# B&R Automation Studio project TrkMster
Automation Studio 4.7.5.60 SP; technology packages: mappMotion 5.12.0, mappView 5.12.0

## Configuration Config1

CPU PC_any, AutomationRuntime C4.72, Build 6.3.0, Safety 0.0, Vc V4.72.0

### Task classes (Cpu.sw)
```
Cyclic#1 (cycle 800 us, tolerance 1600 us):
  TrakMain <- Source.Trak.TrakMain.prg
Cyclic#4:
  Version <- Source.Support.Version.Version.prg
  MachineInf <- Source.Support.MachineInfo.prg
Cyclic#8 (cycle 800 us):
  Program <- Source.Program.prg
DataObjects: McAcpSys
Binaries: FWRules, McAcpSim, arcoal, arsvcreg, TCData, McAcpDrv, mvLoader, arflatprv, udbdef, iomap, Config_1, arconfig, asfw, ashwac, sysconf, User, Role, ashwd, Config_2
Libraries: AsBrStr, McBase, McAxis, McAcpTrak, MpBase, powerlnk, asieccon, sys_lib, arssl, TrkMst, snprintf, LoggingLib, astime, runtime, asstring, ArEventLog, AsTCP, FileIO, brdkSTR
```

### Hardware
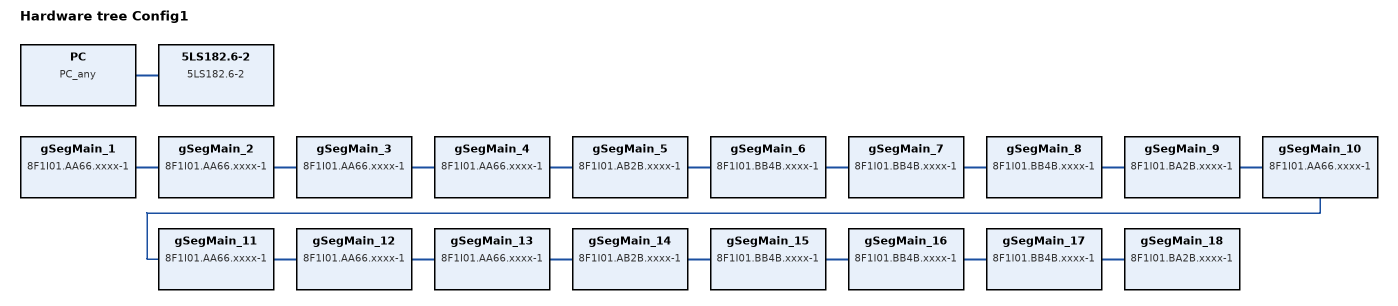
```
5LS182.6-2 : 5LS182.6-2 v1.7.0.0  [SL -> PC.SL1]
PC : PC_any v1.1.0.0 (OrderNumber=PC)
  ConfigurationID = TrkMster_Config1
  ConfigVersion = 0.0.1
  ConfigVersion = 0.1
  ConfigVersion = 0.1
  ConfigVersion = 0.1
  ConfigVersion = 0.1
  ConfigVersion = 0.1
  ConfigVersion = 0.1
  SystemTick = 800
  Cyclic1Duration = 800
  Cyclic1Tolerance = 1600
  Cyclic8Duration = 800
  FileDevice1
  FileDeviceName1 = SvgData
  FileDevicePath1 = ../../../../Logical/SceneViewer/Generated
  ActivateOpcUa = 1
  OpcUaInformationModels_PV_Version = 1
gSegMain_1 : 8F1I01.AA66.xxxx-1 v1.0.0.2  [PLK2 -> gSegMain_2.PLK1 (NodeNumber=1) [Cable Type=PowerlinkCable, Length=10, Version=1.0.0.3]; PLK3 -> 5LS182.6-2.IF1 (NodeNumber=1) [Cable Type=PowerlinkCable, Length=10, Version=1.0.0.3]]
  DriveConfiguration:
    McTypeID = LLMConfig
  DriveConfiguration/Segment:
    Shape = STRAIGHT660
    SegmentReference = gSegMain_1
    StopReaction = UseAssemblySetting
    SpeedFilter = UseAssemblySetting
gSegMain_10 : 8F1I01.AA66.xxxx-1 v1.0.0.2  [PLK1 -> gSegMain_9.PLK2 [Cable Type=PowerlinkCable, Length=10, Version=1.0.0.3]; PLK2 -> gSegMain_11.PLK1 [Cable Type=PowerlinkCable, Length=10, Version=1.0.0.3]]
  DriveConfiguration:
    McTypeID = LLMConfig
  DriveConfiguration/Segment:
    Shape = STRAIGHT660
    SegmentReference = gSegMain_10
    StopReaction = UseAssemblySetting
    SpeedFilter = UseAssemblySetting
gSegMain_11 : 8F1I01.AA66.xxxx-1 v1.0.0.2  [PLK1 -> gSegMain_10.PLK2 [Cable Type=PowerlinkCable, Length=10, Version=1.0.0.3]; PLK2 -> gSegMain_12.PLK1 [Cable Type=PowerlinkCable, Length=10, Version=1.0.0.3]]
  DriveConfiguration:
    McTypeID = LLMConfig
  DriveConfiguration/Segment:
    Shape = STRAIGHT660
    SegmentReference = gSegMain_11
    StopReaction = UseAssemblySetting
    SpeedFilter = UseAssemblySetting
gSegMain_12 : 8F1I01.AA66.xxxx-1 v1.0.0.2  [PLK1 -> gSegMain_11.PLK2 [Cable Type=PowerlinkCable, Length=10, Version=1.0.0.3]; PLK2 -> gSegMain_13.PLK1 [Cable Type=PowerlinkCable, Length=10, Version=1.0.0.3]]
  DriveConfiguration:
    McTypeID = LLMConfig
  DriveConfiguration/Segment:
    Shape = STRAIGHT660
    SegmentReference = gSegMain_12
    StopReaction = UseAssemblySetting
    SpeedFilter = UseAssemblySetting
gSegMain_13 : 8F1I01.AA66.xxxx-1 v1.0.0.2  [PLK1 -> gSegMain_12.PLK2 [Cable Type=PowerlinkCable, Length=10, Version=1.0.0.3]; PLK2 -> gSegMain_14.PLK1 [Cable Type=PowerlinkCable, Length=10, Version=1.0.0.3]]
  DriveConfiguration:
    McTypeID = LLMConfig
  DriveConfiguration/Segment:
    Shape = STRAIGHT660
    SegmentReference = gSegMain_13
    StopReaction = UseAssemblySetting
    SpeedFilter = UseAssemblySetting
gSegMain_14 : 8F1I01.AB2B.xxxx-1 v1.0.0.2  [PLK1 -> gSegMain_13.PLK2 [Cable Type=PowerlinkCable, Length=10, Version=1.0.0.3]; PLK2 -> gSegMain_15.PLK1 [Cable Type=PowerlinkCable, Length=10, Version=1.0.0.3]]
  DriveConfiguration:
    McTypeID = LLMConfig
  DriveConfiguration/Segment:
    Shape = STRAIGHT105_TO_CIRCULAR
    SegmentReference = gSegMain_14
    StopReaction = UseAssemblySetting
    SpeedFilter = UseAssemblySetting
gSegMain_15 : 8F1I01.BB4B.xxxx-1 v1.0.0.2  [PLK1 -> gSegMain_14.PLK2 [Cable Type=PowerlinkCable, Length=10, Version=1.0.0.3]; PLK2 -> gSegMain_16.PLK1 [Cable Type=PowerlinkCable, Length=10, Version=1.0.0.3]]
  DriveConfiguration:
    McTypeID = LLMConfig
  DriveConfiguration/Segment:
    Shape = CIRCULAR
    SegmentReference = gSegMain_15
    StopReaction = UseAssemblySetting
    SpeedFilter = UseAssemblySetting
gSegMain_16 : 8F1I01.BB4B.xxxx-1 v1.0.0.2  [PLK1 -> gSegMain_15.PLK2 [Cable Type=PowerlinkCable, Length=10, Version=1.0.0.3]; PLK2 -> gSegMain_17.PLK1 [Cable Type=PowerlinkCable, Length=10, Version=1.0.0.3]]
  DriveConfiguration:
    McTypeID = LLMConfig
  DriveConfiguration/Segment:
    Shape = CIRCULAR
    SegmentReference = gSegMain_16
    StopReaction = UseAssemblySetting
    SpeedFilter = UseAssemblySetting
gSegMain_17 : 8F1I01.BB4B.xxxx-1 v1.0.0.2  [PLK1 -> gSegMain_16.PLK2 [Cable Type=PowerlinkCable, Length=10, Version=1.0.0.3]; PLK2 -> gSegMain_18.PLK1 [Cable Type=PowerlinkCable, Length=10, Version=1.0.0.3]]
  DriveConfiguration:
    McTypeID = LLMConfig
  DriveConfiguration/Segment:
    Shape = CIRCULAR
    SegmentReference = gSegMain_17
    StopReaction = UseAssemblySetting
    SpeedFilter = UseAssemblySetting
gSegMain_18 : 8F1I01.BA2B.xxxx-1 v1.0.0.2  [PLK1 -> gSegMain_17.PLK2 [Cable Type=PowerlinkCable, Length=10, Version=1.0.0.3]]
  DriveConfiguration:
    McTypeID = LLMConfig
  DriveConfiguration/Segment:
    Shape = CIRCULAR_TO_STRAIGHT105
    SegmentReference = gSegMain_18
    StopReaction = UseAssemblySetting
    SpeedFilter = UseAssemblySetting
gSegMain_2 : 8F1I01.AA66.xxxx-1 v1.0.0.2  [PLK1 -> gSegMain_1.PLK2 [Cable Type=PowerlinkCable, Length=10, Version=1.0.0.3]; PLK2 -> gSegMain_3.PLK1 [Cable Type=PowerlinkCable, Length=10, Version=1.0.0.3]]
  DriveConfiguration:
    McTypeID = LLMConfig
  DriveConfiguration/Segment:
    Shape = STRAIGHT660
    SegmentReference = gSegMain_2
    StopReaction = UseAssemblySetting
    SpeedFilter = UseAssemblySetting
gSegMain_3 : 8F1I01.AA66.xxxx-1 v1.0.0.2  [PLK1 -> gSegMain_2.PLK2 [Cable Type=PowerlinkCable, Length=10, Version=1.0.0.3]; PLK2 -> gSegMain_4.PLK1 [Cable Type=PowerlinkCable, Length=10, Version=1.0.0.3]]
  DriveConfiguration:
    McTypeID = LLMConfig
  DriveConfiguration/Segment:
    Shape = STRAIGHT660
    SegmentReference = gSegMain_3
    StopReaction = UseAssemblySetting
    SpeedFilter = UseAssemblySetting
gSegMain_4 : 8F1I01.AA66.xxxx-1 v1.0.0.2  [PLK1 -> gSegMain_3.PLK2 [Cable Type=PowerlinkCable, Length=10, Version=1.0.0.3]; PLK2 -> gSegMain_5.PLK1 [Cable Type=PowerlinkCable, Length=10, Version=1.0.0.3]]
  DriveConfiguration:
    McTypeID = LLMConfig
  DriveConfiguration/Segment:
    Shape = STRAIGHT660
    SegmentReference = gSegMain_4
    StopReaction = UseAssemblySetting
    SpeedFilter = UseAssemblySetting
gSegMain_5 : 8F1I01.AB2B.xxxx-1 v1.0.0.2  [PLK1 -> gSegMain_4.PLK2 [Cable Type=PowerlinkCable, Length=10, Version=1.0.0.3]; PLK2 -> gSegMain_6.PLK1 [Cable Type=PowerlinkCable, Length=10, Version=1.0.0.3]]
  DriveConfiguration:
    McTypeID = LLMConfig
  DriveConfiguration/Segment:
    Shape = STRAIGHT105_TO_CIRCULAR
    SegmentReference = gSegMain_5
    StopReaction = UseAssemblySetting
    SpeedFilter = UseAssemblySetting
gSegMain_6 : 8F1I01.BB4B.xxxx-1 v1.0.0.2  [PLK1 -> gSegMain_5.PLK2 [Cable Type=PowerlinkCable, Length=10, Version=1.0.0.3]; PLK2 -> gSegMain_7.PLK1 [Cable Type=PowerlinkCable, Length=10, Version=1.0.0.3]]
  DriveConfiguration:
    McTypeID = LLMConfig
  DriveConfiguration/Segment:
    Shape = CIRCULAR
    SegmentReference = gSegMain_6
    StopReaction = UseAssemblySetting
    SpeedFilter = UseAssemblySetting
gSegMain_7 : 8F1I01.BB4B.xxxx-1 v1.0.0.2  [PLK1 -> gSegMain_6.PLK2 [Cable Type=PowerlinkCable, Length=10, Version=1.0.0.3]; PLK2 -> gSegMain_8.PLK1 [Cable Type=PowerlinkCable, Length=10, Version=1.0.0.3]]
  DriveConfiguration:
    McTypeID = LLMConfig
  DriveConfiguration/Segment:
    Shape = CIRCULAR
    SegmentReference = gSegMain_7
    StopReaction = UseAssemblySetting
    SpeedFilter = UseAssemblySetting
gSegMain_8 : 8F1I01.BB4B.xxxx-1 v1.0.0.2  [PLK1 -> gSegMain_7.PLK2 [Cable Type=PowerlinkCable, Length=10, Version=1.0.0.3]; PLK2 -> gSegMain_9.PLK1 [Cable Type=PowerlinkCable, Length=10, Version=1.0.0.3]]
  DriveConfiguration:
    McTypeID = LLMConfig
  DriveConfiguration/Segment:
    Shape = CIRCULAR
    SegmentReference = gSegMain_8
    StopReaction = UseAssemblySetting
    SpeedFilter = UseAssemblySetting
gSegMain_9 : 8F1I01.BA2B.xxxx-1 v1.0.0.2  [PLK1 -> gSegMain_8.PLK2 [Cable Type=PowerlinkCable, Length=10, Version=1.0.0.3]; PLK2 -> gSegMain_10.PLK1 [Cable Type=PowerlinkCable, Length=10, Version=1.0.0.3]]
  DriveConfiguration:
    McTypeID = LLMConfig
  DriveConfiguration/Segment:
    Shape = CIRCULAR_TO_STRAIGHT105
    SegmentReference = gSegMain_9
    StopReaction = UseAssemblySetting
    SpeedFilter = UseAssemblySetting
```

### Config_1.assembly - PC/mappMotion/Config_1.assembly
```
Element gAssembly_1 (Type=assembly)
  Tracks:
    TrackSeparation = 0.030
    Track[1]:
      Segments:
        SegmentRef[1] = ::gSegMain_1
        SegmentRef[2] = ::gSegMain_2
        SegmentRef[3] = ::gSegMain_3
        SegmentRef[4] = ::gSegMain_4
        SegmentRef[5] = ::gSegMain_5
        SegmentRef[6] = ::gSegMain_6
        SegmentRef[7] = ::gSegMain_7
        SegmentRef[8] = ::gSegMain_8
        SegmentRef[9] = ::gSegMain_9
        SegmentRef[10] = ::gSegMain_10
        SegmentRef[11] = ::gSegMain_11
        SegmentRef[12] = ::gSegMain_12
        SegmentRef[13] = ::gSegMain_13
        SegmentRef[14] = ::gSegMain_14
        SegmentRef[15] = ::gSegMain_15
        SegmentRef[16] = ::gSegMain_16
        SegmentRef[17] = ::gSegMain_17
        SegmentRef[18] = ::gSegMain_18
      Position = Absolute
        SegmentRef = ::gSegMain_1
        SegmentCountDirection = RightToLeft
        Translation:
          X = 0.0
          Y = 0.0
          Z = 0.0
        Orientation:
          Angle1 = 0.0
          Angle2 = 0.0
          Angle3 = 0.0
  CommonSegmentSettings:
    SegmentSimulationOnPLC = Off
    StopReaction = InductionHalt
    SpeedFilter = NotUsed
    ControllerParameters:
      DefaultParameter:
        Controller:
          Position:
            ProportionalGain = 0.0
          Speed:
            ProportionalGain = 0.0
            IntegrationTime = 0.0
          FeedForward:
            TotalMass = 0.0
            ForcePositive = 0.0
            ForceNegative = 0.0
            SpeedForceFactor = 0.0
            ForceLoad = 0.0
        MovementErrorLimits:
          PositionError = 0.0
          VelocityError = 0.0
      AdditionalParameterSets = NotUsed
    ShuttleIdentificationTime = 0
  Shuttles:
    MaxShuttleCount = 10
    DistanceReserve:
      Collision = 0.002
      ErrorStop = 0.006
    ShuttleStereotypes:
      ShuttleStRef[1] = ShuttleStereotype_1
    MagnetPlateConfigurations:
      ShuttleType[1] = 8F1SA.100.xxxxxx-x
    CollisionAvoidance:
      Strategy = Constant
      MaximumModelDimensions:
        Length:
          ExtentToFront = 0.025
          ExtentToBack = 0.025
        Width:
          Width = 0.046
  Visualization:
    MonitoringPv = ::gShuttleMon
    ProcessingTaskClass = 1
```

### Config_2.shuttlestereotype - PC/mappMotion/Config_2.shuttlestereotype
```
Element ShuttleStereotype_1 (Type=shuttlestereotype)
  MeasurementUnit = 5067858
  MeasurementResolution = 0.00001
  MovementLimits = Internal
    VelocityIsReadOnly = 0
    Velocity:
      Velocity = 4.0
    AccelerationIsReadOnly = 0
    Acceleration:
      Acceleration = 10.0
    DecelerationIsReadOnly = 0
    Deceleration:
      Deceleration = 10.0
  JerkFilter = Used
    JerkTime = 0.02
  UserData:
    Size = 3
```

### Config_3.sector - PC/mappMotion/Config_3.sector
```
Element secMain (Type=sector)
  Type = Composed
    StartSegment:
      SegmentRef = ::gSegMain_1
    IntermediateSegments:
      SegmentRef[1] = ::gSegMain_2
      SegmentRef[2] = ::gSegMain_3
      SegmentRef[3] = ::gSegMain_4
      SegmentRef[4] = ::gSegMain_5
      SegmentRef[5] = ::gSegMain_6
      SegmentRef[6] = ::gSegMain_7
      SegmentRef[7] = ::gSegMain_8
      SegmentRef[8] = ::gSegMain_9
      SegmentRef[9] = ::gSegMain_10
      SegmentRef[10] = ::gSegMain_11
      SegmentRef[11] = ::gSegMain_12
      SegmentRef[12] = ::gSegMain_13
      SegmentRef[13] = ::gSegMain_14
      SegmentRef[14] = ::gSegMain_15
      SegmentRef[15] = ::gSegMain_16
      SegmentRef[16] = ::gSegMain_17
    EndSegment:
      SegmentRef = ::gSegMain_18
      PositionRelativeTo = FromEnd
```

## Logical view

Binary libraries used (declarations not repeated): operator, runtime, astime, AsIecCon, AsBrStr, McBase 5.12.0, McAxis 5.12.0, McAcpTrak 5.12.0, MpBase 5.12.0, snprintf 1.10.2, LoggingLib 2.30.1, asstring, ArEventLog, AsTCP, FileIO

### Global.typ - Global data types
```iecst
TYPE
	UserDataTyp : 	STRUCT
		Red : USINT;
		Green : USINT;
		Blue : USINT;
	END_STRUCT;
END_TYPE
```

### Global.var - Global variables
```iecst
VAR
	gShuttleMon : McAcpTrakAssemblyMonData;
	gPowered : BOOL;
END_VAR
```

### Segments.var - Global variables
```iecst
VAR
	gSegMain_1 : McSegmentType;
	gSegMain_2 : McSegmentType;
	gSegMain_3 : McSegmentType;
	gSegMain_4 : McSegmentType;
	gSegMain_5 : McSegmentType;
	gSegMain_6 : McSegmentType;
	gSegMain_7 : McSegmentType;
	gSegMain_8 : McSegmentType;
	gSegMain_9 : McSegmentType;
	gSegMain_10 : McSegmentType;
	gSegMain_11 : McSegmentType;
	gSegMain_12 : McSegmentType;
	gSegMain_13 : McSegmentType;
	gSegMain_14 : McSegmentType;
	gSegMain_15 : McSegmentType;
	gSegMain_16 : McSegmentType;
	gSegMain_17 : McSegmentType;
END_VAR
```

### Package Logical/Libraries - Global libraries

- Library Logical/Libraries/brdkSTR (ANSIC, version 1.03.1) (no source held here)

### Library Logical/Libraries/TrkMst (ANSIC)
Depends on: McAcpTrak, snprintf, brdkSTR

#### Types.typ - Exported data types
```iecst
(*Track Master Core Types*)

TYPE
	tmCoreInternalTyp : 	STRUCT  (*Internal Datatype*)
		TypeID : UDINT; (*TypeID to help with handle application*)
		State : USINT; (*State of execution*)
		Axes : ARRAY[0..tmMAX_SHUTLE_ARRAY]OF tmCoreAxisLookupTyp; (*Axis Lookup table based on the current Shuttle Index*)
		Fbs : tmCoreFbTyps; (*Internal Function blocks*)
		ShCount : USINT; (*Shuttle Count*)
	END_STRUCT;
	tmCoreViewBoxCfgTyp : 	STRUCT  (*Attributes of the SVG's viewbox*)
		MinX : REAL; (*Minimum x position*)
		MinY : REAL; (*minimum y position*)
		Width : REAL; (*Width of viewbox*)
		Height : REAL; (*Height of viewbox*)
	END_STRUCT;
	tmCoreStateEnum :
		( (*State of execution*)
		tmCORE_OFF, (*Waiting for enable command*)
		tmCORE_INIT, (*Initialization state*)
		tmCORE_GET_SH, (*Get the shuttle in the assembly*)
		tmCORE_GET_NEXT, (*Set the next command*)
		tmCORE_RUNNING, (*Running state*)
		tmCORE_RESET, (*Resetting state*)
		tmCORE_ERROR (*Error state*)
		);
	tmCoreErrorEnum :
		( (*Error Enumeration*)
		tmCORE_ERR_OK := 0, (*No error present*)
		tmCORE_ERR_INVALID_ASSEMBLY := -61000, (*Invalid input assembly reference*)
		tmCORE_ERR_SH_COUNT_EXCEEDED := -61001, (*Maximum shuttle count exceeded. Need to increase max shuttle count constant*)
		tmCORE_ERR_STR_LEN_EXCEEDED := -61002 (*The built string is too long, need to increase the maximum size to prevent page faulting*)
		);
	tmCoreSvgLengthsTyp : 	STRUCT  (*String lengths of SVGs*)
		ContentLength : UDINT; (*String Length of SVG Content string*)
		TransformLength : UDINT; (*String Length of SVG Transform string*)
	END_STRUCT;
	tmCoreFbTyps : 	STRUCT  (*Internal Function blocks*)
		AsmGetShuttle : MC_BR_AsmGetShuttle_AcpTrak;
	END_STRUCT;
	tmCoreAxisLookupTyp : 	STRUCT  (*Lookup table datatype*)
		Present : BOOL; (*Axis is present and a valid reference exists*)
		Axis : McAxisType; (*Axis information*)
	END_STRUCT;
	tmCoreOptionsTyp : 	STRUCT  (*Options for Core Function Block*)
		Color : tmCoreColorOptionTyp; (*Shuttle Color Option*)
	END_STRUCT;
	tmCoreColorOptionTyp : 	STRUCT  (*Shuttle Color Option*)
		Enabled : BOOL; (*Option is enabled*)
		Offsets : tmCoreColorOffsetsTyp; (*Userdata color offsets*)
	END_STRUCT;
	tmCoreColorOffsetsTyp : 	STRUCT  (*Userdata color offsets*)
		Red : UDINT; (*Offset for UserData address for the Red color in USINT*)
		Green : UDINT; (*Offset for UserData address for the Green color in USINT*)
		Blue : UDINT; (*Offset for UserData address for the Blue color in USINT*)
	END_STRUCT;
END_TYPE

(*Track Master Shuttle Control Types*)

TYPE
	tmShuttleControlParsTyp : 	STRUCT  (*Input parameters for Shuttle Control*)
		Position : LREAL; (*Destination position for Absolute and Velocity commands*)
		Distance : LREAL; (*Distance for all relative commands*)
		Vel : REAL; (*Comanded Movement velocity*)
		Accel : REAL; (*Comanded Movement acceleration*)
		Decel : REAL; (*Comanded Movement deceleration*)
	END_STRUCT;
	tmShuttleControlInternalTyp : 	STRUCT  (*Internal data type*)
		State : tmShuttleControlStatesEnum; (*State of execution*)
		CoreInt : REFERENCE TO tmCoreInternalTyp; (*Internal data for the Core function block*)
		CurrentAxis : McAxisType; (*Current selected Axis*)
		Fbs : tmShuttleControlFbTyp; (*Internal function blocks*)
		Idx : USINT; (*Selected Index for the axis lookup table*)
		LastIdx : USINT; (*Last cycle selected index for the axis lookup table*)
	END_STRUCT;
	tmShuttleControlFbTyp : 	STRUCT  (*Internal Function Blocks*)
		ShGetInfo : MC_BR_ShReadInfo_AcpTrak; (*Shuttle Get info*)
		ElMoveAbs : MC_BR_ElasticMoveAbs_AcpTrak; (*Elastic move absolute command*)
		ElMoveAdd : MC_BR_ElasticMoveAdd_AcpTrak; (*Elastic move addtive command*)
	END_STRUCT;
	tmShuttleControlErrorEnum :
		( (*Error enumeration*)
		tmSH_CONTROL_ERR_OK := 0, (*No error currently*)
		tmSH_CONTROL_WARN_SH_NOT_AVAIL := -52000, (*Shuttle Currently not listed as available*)
		tmSH_CONTROL_WARN_NO_ELEM_FND := -52001, (*Input selected element did not return a shuttle*)
		tmSH_CONTROL_ERR_INVALID_HANDLE := -62000, (*Invalid input handle*)
		tmSH_CONTROL_ERR_EL_MOVE := -62001 (*Error in an elastic movment*)
		);
	tmShuttleControlStatesEnum :
		( (*State of execution*)
		tmSH_CONTROL_OFF, (*Off State*)
		tmSH_CONTROL_INIT, (*Init/Waiting for valid ShElement state*)
		tmSH_CONTROL_IDLE, (*Idle waiting for a command state*)
		tmSH_CONTROL_EL_MOVE_ABS, (*Move Elastic absoulte active state*)
		tmSH_CONTROL_EL_MOVE_ADD, (*Move Elastic Additive active state*)
		tmSH_CONTROL_MOVE_DONE, (*Move has completed*)
		tmSH_CONTROL_ERROR (*Error present on the FB*)
		);
END_TYPE
```

#### Constants.var - Exported constants
```iecst
VAR CONSTANT
	tmMAX_SHUTTLE_COUNT : USINT := 150;
	tmMAX_SHUTLE_ARRAY : USINT := tmMAX_SHUTTLE_COUNT-1;
	tmCORE_CORE_TYPE_ID : DINT := 651684313;
	tmCORE_MAX_STR_LEN : UDINT := 3000;
END_VAR
```

#### TrkMst.fun - Exported functions and function blocks
```iecst
FUNCTION_BLOCK tmCore (*Core Track Master Function Block*)
	VAR_INPUT
		Enable : BOOL; (*Enables the core functionality*)
		ErrorRest : BOOL; (*Reset any present errors*)
		Assembly : REFERENCE TO McAssemblyType; (*Assembly reference to monitor*)
		ShuttleMon : REFERENCE TO McAcpTrakAssemblyMonData; (*Shuttle Monitor structure for the assembly*)
		ViewBoxCfg : tmCoreViewBoxCfgTyp; (*View box configuration for the SVG*)
		Options : REFERENCE TO tmCoreOptionsTyp; (*Options for the core fb*)
	END_VAR
	VAR_OUTPUT
		Error : BOOL; (*Error present on FB*)
		ErrorID : tmCoreErrorEnum; (*Error ID of current error*)
		Active : BOOL; (*Function block is active*)
		SvgContent : STRING[tmCORE_MAX_STR_LEN]; (*SVG Content string to tie to a Paper widget*)
		SvgTransform : STRING[tmCORE_MAX_STR_LEN]; (*SVG Transform string to tie to a paper widget*)
		StrLengths : tmCoreSvgLengthsTyp; (*Diagnostic viewer to see current lengths of SVG Content/Transform*)
		Handle : UDINT; (*Handle used for other Track Master Function Blocks*)
	END_VAR
	VAR
		Internal : tmCoreInternalTyp; (*Internal data type*)
	END_VAR
END_FUNCTION_BLOCK

FUNCTION_BLOCK tmShuttleControl (*Shuttle Control Function Block*)
	VAR_INPUT
		Enable : BOOL; (*Enables the shuttle controller*)
		Handle : UDINT; (*Handle of the Core Track Master Function Block*)
		SelectedElem : STRING[80]; (*Selected Element String that is populated from a Paper Widget*)
		ElasticMoveAbs : BOOL; (*Command to send shuttle on Elastic Move Absolute*)
		ElasticMoveAdd : BOOL; (*Command to send shuttle on Elastic Move Additive*)
		Parameters : REFERENCE TO tmShuttleControlParsTyp; (*Parameters for movement commands*)
	END_VAR
	VAR_OUTPUT
		Active : BOOL; (*Function block is currently Active*)
		MovementActive : BOOL; (*Controlled Shuttle is currently moving*)
		MovementDone : BOOL; (*Controlled Shuttle has completed movement*)
		Valid : BOOL; (*Input Selected Element is a valid controllable shuttle*)
		ShInfo : McAcpTrakShInfoType; (*Selected shuttle's current info. Only is Valid when Valid flag is set*)
		Error : BOOL; (*Error Present on FB*)
		ErrorID : DINT; (*Error ID of current Error*)
	END_VAR
	VAR
		Internal : tmShuttleControlInternalTyp; (*Internal data type*)
	END_VAR
END_FUNCTION_BLOCK
```

#### tmCore.c
```c
#include <bur/plctypes.h>

#define TRUE 1
#define FALSE 0

#ifdef __cplusplus
	extern "C"
	{
#endif
#include "TrkMst.h"
#ifdef __cplusplus
	};
#endif
//Verify that the two string lengths do not exceed a length
plcbit CheckStrLen(char* dest,char* source,UDINT length){
	if(brdkStrLen(dest) + brdkStrLen(source) >= length){
		return FALSE;
	}
	else{
		return TRUE;
	}
}
DINT BuildShuttlePolygon(char* dest,
		USINT idx,
		LREAL length,
		LREAL width,
		UDINT userDataAdr,
		struct tmCoreColorOptionTyp* colorOption){

	char tmp[150];
	USINT red,blue,green;
	struct UserDataTyp* tst;

	if(!colorOption->Enabled){
		snprintf2(tmp,150,"<polygon id=\"sh%d\" points=\"0,0 %0f,0 , %f,%f %f,%f 0,%f\" style=\"fill:rgb(0,255,0);\"/>",
			idx,	//polygon index
			(length-width/2.0),//p1.x
			length,	//p1.y
			width/2.0, //p2.x
			(length-width/2.0),//p2.y
			width,//p2.x
			width); //p3.y
	}
	else{
		brsmemcpy(&red,userDataAdr + colorOption->Offsets.Red,sizeof(USINT));
		brsmemcpy(&green,userDataAdr + colorOption->Offsets.Green,sizeof(USINT));
		brsmemcpy(&blue,userDataAdr + colorOption->Offsets.Blue,sizeof(USINT));

		snprintf2(tmp,150,"<polygon id=\"sh%d\" points=\"0,0 %0f,0 , %f,%f %f,%f 0,%f\" style=\"fill:rgb(%d,%d,%d);\"/>",
			idx,	//polygon index
			(length-width/2.0),//p1.x
			length,	//p1.y
			width/2.0, //p2.x
			(length-width/2.0),//p2.y
			width,//p2.x
			width,
			red,
			green,
			blue); //p3.y
	}
	if(CheckStrLen(dest,&tmp,tmCORE_MAX_STR_LEN)){
		brsstrcat(dest,&tmp);
		return tmCORE_ERR_OK;
	}
	else
		return tmCORE_ERR_STR_LEN_EXCEEDED;
}

//This function loops through the assembly monitor data and builds a SVG string + SVG Transform. Will return 0 if succesful
//Will monitor to make sure the string lengths are not exceeded
DINT BuildStrings(struct McAcpTrakAssemblyMonData* mon,
		char* svgContent,char* svgTransform,
		struct tmCoreViewBoxCfgTyp* viewBox,
		struct tmCoreOptionsTyp* coreOptions){
	USINT i;
	USINT transCounter;
	transCounter = 0;
	char tmp[150];
	brsmemset(svgContent,0,sizeof(svgContent));
	brsmemset(svgTransform,0,sizeof(svgTransform));

	snprintf2(tmp,150,"<svg viewBox=\"%f %f %f %f\">",
		viewBox->MinX,
		viewBox->MinY,
		viewBox->Width,
		viewBox->Height);
	if(CheckStrLen(svgContent,&tmp,tmCORE_MAX_STR_LEN)){
		brsstrcat(svgContent,&tmp);
	}
	else
		return tmCORE_ERR_STR_LEN_EXCEEDED;
	brsstrcat(svgTransform,&"[");

	for (i = 0; i < tmMAX_SHUTTLE_COUNT; i++){
		if(mon->Shuttle[i].Available){
			brsmemset(&tmp,0,sizeof(tmp));

			LREAL width;
			LREAL length;
			LREAL shCenterX;
			LREAL shCenterY;

			width = mon->Shuttle[i].Width / 1000.0;
			length = (mon->Shuttle[i].ExtentToBack + mon->Shuttle[i].ExtentToFront)/ 1000.0;
			shCenterX = mon->Shuttle[i].Position.X / 1000.0 - mon->Shuttle[i].ExtentToBack / 1000.0;
			shCenterY = -(mon->Shuttle[i].Position.Y / 1000.0 + width / 2.0);

			snprintf2(tmp,150,"<g id=\"Shuttle%d\">",mon->Shuttle[i].Index);
			if(CheckStrLen(svgContent,&tmp,tmCORE_MAX_STR_LEN)){
				brsstrcat(svgContent,&tmp);
			}
			else
				return tmCORE_ERR_STR_LEN_EXCEEDED;

			DINT returnVal;
			returnVal = BuildShuttlePolygon(svgContent,mon->Shuttle[i].Index,length,width,mon->Shuttle[i].UserData,&coreOptions->Color);
			if(returnVal!= tmCORE_ERR_OK)
				return returnVal;

			snprintf2(tmp,150,"<text x=\"%f\" y=\"%f\" font-weight=\"bold\" font-size=\"0.035px\">%d</text>",
				mon->Shuttle[i].ExtentToBack / 2000.0,
				width * 3.0 / 4.0,
				mon->Shuttle[i].Index);
			if(CheckStrLen(svgContent,&tmp,tmCORE_MAX_STR_LEN)){
				brsstrcat(svgContent,&tmp);
			}
			else
				return tmCORE_ERR_STR_LEN_EXCEEDED;

			//Create an invisible bounding rectangle to handle the click event. "Invisible" by using the alpha channel, if you use the
			//Vibisility property, the click event will not fire for the SVG
			snprintf2(tmp,150,"<rect id=\"ID%d\" width=\"%f\" height=\"%f\" style=\"fill:rgba(0,0,0,0)\"/>",
				mon->Shuttle[i].Index,
				length,
				width);
			if(CheckStrLen(svgContent,&tmp,tmCORE_MAX_STR_LEN)){
				brsstrcat(svgContent,&tmp);
			}
			else
				return tmCORE_ERR_STR_LEN_EXCEEDED;

			if(CheckStrLen(svgContent,&"</g>",tmCORE_MAX_STR_LEN)){
				brsstrcat(svgContent,&"</g>");
			}
			else
				return tmCORE_ERR_STR_LEN_EXCEEDED;

			//Check to see if we've had more transforms to add a comma between the units
			if(transCounter>0){
				if(CheckStrLen(svgTransform,&",",tmCORE_MAX_STR_LEN)){
					brsstrcat(svgTransform,&",");
				}
				else
					return tmCORE_ERR_STR_LEN_EXCEEDED;
			}
			//Preform translation
			snprintf2(tmp,150,"{\"select\":\"#Shuttle%d\",\"duration\":100,\"display\":true,\"translate\":[%f,%f]},",
				mon->Shuttle[i].Index,
				shCenterX,
				shCenterY,
				-mon->Shuttle[i].Orientation.Angle1,
				length/2.0,
				width/2.0);
			if(CheckStrLen(svgTransform,&tmp,tmCORE_MAX_STR_LEN)){
				brsstrcat(svgTransform,&tmp);
			}
			else
				return tmCORE_ERR_STR_LEN_EXCEEDED;
			//Preform rotation
			snprintf2(tmp,150,"{\"select\":\"#sh%d\",\"duration\":100,\"display\":true,\"spin\":[%f,%f,%f]}",
				mon->Shuttle[i].Index,
				-mon->Shuttle[i].Orientation.Angle1, //Spin amount
				length/2.0,	//Spin center x
				width/2.0); //Spin center y
			if(CheckStrLen(svgTransform,&tmp,tmCORE_MAX_STR_LEN)){
				brsstrcat(svgTransform,&tmp);
			}
			else
				return tmCORE_ERR_STR_LEN_EXCEEDED;
			transCounter++;
		}

	}
	if(CheckStrLen(svgContent,&"</svg>",tmCORE_MAX_STR_LEN)){
		brsstrcat(svgContent,&"</svg>");
	}
	else
		return tmCORE_ERR_STR_LEN_EXCEEDED;
	if(CheckStrLen(svgTransform,&"]",tmCORE_MAX_STR_LEN)){
		brsstrcat(svgTransform,&"]");
	}
	else
		return tmCORE_ERR_STR_LEN_EXCEEDED;

	//No Error, finished everything return OK
	return tmCORE_ERR_OK;
}

/* Core Track Master function blocks. Handles the building of the SVG string */
void tmCore(struct tmCore* inst)
{
	switch (inst->Internal.State){
		case tmCORE_OFF:
			//******************************************************************************** Off state
			if(inst->Enable){
				inst->Internal.TypeID = tmCORE_CORE_TYPE_ID;
				inst->Handle = &inst->Internal;

				inst->Internal.Fbs.AsmGetShuttle.Assembly = inst->Assembly;
				inst->Internal.Fbs.AsmGetShuttle.Enable = TRUE;
				inst->Active = TRUE;
				inst->Internal.State = tmCORE_INIT;
			}
			break;
		case tmCORE_INIT:
			//Reset the lookup array just for safety
			brsmemset(&inst->Internal.Axes,0,sizeof(inst->Internal.Axes));

        	inst->Internal.State = tmCORE_GET_SH;
			break;
		case tmCORE_GET_SH:
			//******************************************************************************** Get Shuttle state
			if(inst->Internal.Fbs.AsmGetShuttle.Error){
				inst->Error = TRUE;
				inst->ErrorID = tmCORE_ERR_INVALID_ASSEMBLY;

				inst->Internal.State = tmCORE_ERROR;
			}
			else if(inst->Internal.Fbs.AsmGetShuttle.Valid){
				if(inst->Internal.Fbs.AsmGetShuttle.TotalCount >= tmMAX_SHUTTLE_COUNT
				|| inst->Internal.Fbs.AsmGetShuttle.AdditionalInfo.ShuttleID >= tmMAX_SHUTTLE_COUNT){

					inst->Error = TRUE;
					inst->ErrorID = tmCORE_ERR_SH_COUNT_EXCEEDED;

					inst->Internal.State = tmCORE_ERROR;
				}
				else{
					inst->Internal.Axes[inst->Internal.Fbs.AsmGetShuttle.AdditionalInfo.ShuttleID].Present = TRUE;
					inst->Internal.Axes[inst->Internal.Fbs.AsmGetShuttle.AdditionalInfo.ShuttleID].Axis = inst->Internal.Fbs.AsmGetShuttle.Axis;
					inst->Internal.Fbs.AsmGetShuttle.Next = FALSE;

					if(inst->Internal.Fbs.AsmGetShuttle.RemainingCount == 0){
						//Done populating the lookup array, moving on
						inst->Internal.Fbs.AsmGetShuttle.Enable = FALSE;

						inst->Internal.State = tmCORE_RUNNING;
					}
					else{
						inst->Internal.ShCount++;

						inst->Internal.State = tmCORE_GET_NEXT;
					}
				}
			}
			break;
		case tmCORE_GET_NEXT:
			//******************************************************************************** Get next shuttle state
			inst->Internal.Fbs.AsmGetShuttle.Next = TRUE;
			inst->Internal.State = tmCORE_GET_SH;
			break;
		case tmCORE_RUNNING:
			inst->ErrorID = BuildStrings(inst->ShuttleMon,&inst->SvgContent,&inst->SvgTransform,&inst->ViewBoxCfg,inst->Options);
			inst->StrLengths.ContentLength = brdkStrLen(&inst->SvgContent);
			inst->StrLengths.TransformLength = brdkStrLen(&inst->SvgTransform);

			if(inst->ErrorID != tmCORE_ERR_OK){
				inst->Error = TRUE;

				inst->Internal.State = tmCORE_ERROR;
			}
			break;
		case tmCORE_RESET:
        	//Try and recover by resetting any blocks

			break;
		case tmCORE_ERROR:
			if(inst->ErrorRest){
				inst->Error = FALSE;
				inst->ErrorID = tmCORE_ERR_OK;

				inst->Internal.State = tmCORE_OFF;
			}
			break;
	}
	//FB calls
	MC_BR_AsmGetShuttle_AcpTrak(&inst->Internal.Fbs.AsmGetShuttle);
}
```

#### tmShuttleControl.c
```c
#include <bur/plctypes.h>

#define TRUE 1
#define FALSE 0

#ifdef __cplusplus
	extern "C"
	{
#endif
#include "TrkMst.h"
#ifdef __cplusplus
	};
#endif

plcbit CheckValidity(char* selectedElem){
	char buf[2];
	//Get a substring of the first 3 characters
	brdkStrSubStr(&buf,selectedElem,0,3);
	//Look at the start of the selectedID, if it starts with #ID then we know a shuttle has been clicked
	if(0 == brsstrcmp(&buf,&"#ID")){
		return TRUE;
	}
	else{
		return FALSE;
	}
}
USINT GetIndex(char* selectedElem){
	char buf[3];
	brdkStrSubStr(&buf,selectedElem,3,brdkStrLen(selectedElem) - 3);
	return (USINT)brdkStrAToUdint(&buf,BRDK_STR_CONVERT_DECIMAL);
}
/* Function block for handling a shuttle control provided from the paper element's selected element ID. Must be paired with the tmCore FB */
void tmShuttleControl(struct tmShuttleControl* inst)
{
	if(inst->Valid){
		inst->ShInfo = inst->Internal.Fbs.ShGetInfo.ShuttleInfo;
	}
	switch (inst->Internal.State){
		case tmSH_CONTROL_OFF:
			//******************************************************************************** Off state
			if(inst->Enable){
				if(inst->Handle == 0){
					inst->Error = TRUE;
					inst->ErrorID = tmSH_CONTROL_ERR_INVALID_HANDLE;

					inst->Internal.State = tmSH_CONTROL_ERROR;
				}
				else{
					inst->Internal.CoreInt = (tmCoreInternalTyp*)inst->Handle;
					if(inst->Internal.CoreInt->TypeID != tmCORE_CORE_TYPE_ID){
						inst->Error = TRUE;
						inst->ErrorID = tmSH_CONTROL_ERR_INVALID_HANDLE;

						inst->Internal.State = tmSH_CONTROL_ERROR;
					}
					else{
						inst->Active = TRUE;

						inst->Internal.State = tmSH_CONTROL_INIT;
					}
				}
			}
			break;
		case tmSH_CONTROL_INIT:
			//******************************************************************************** Init state
			if(CheckValidity(&inst->SelectedElem)){	//Checking for the validity of the selected element format
				inst->Internal.Idx = GetIndex(&inst->SelectedElem);	//Pulling the index from the string
				if(inst->Internal.CoreInt->Axes[inst->Internal.Idx].Present){ //Verifying that index has a valid access in it
					inst->ErrorID = tmSH_CONTROL_ERR_OK;
					inst->Valid = TRUE;
					inst->Internal.CurrentAxis = inst->Internal.CoreInt->Axes[inst->Internal.Idx].Axis;

					inst->Internal.Fbs.ShGetInfo.Axis = &inst->Internal.CurrentAxis;
					inst->Internal.Fbs.ShGetInfo.Enable = TRUE;

					inst->Internal.State = tmSH_CONTROL_IDLE;
				}
				else{
					inst->ErrorID = tmSH_CONTROL_WARN_SH_NOT_AVAIL;
				}
			}
			else{
				inst->ErrorID = tmSH_CONTROL_WARN_NO_ELEM_FND;
			}

			break;
		case tmSH_CONTROL_IDLE:
			//******************************************************************************** Get Shuttle state
			//Need to check for if the selected element has changed
			inst->Internal.LastIdx = inst->Internal.Idx;
			if(CheckValidity(&inst->SelectedElem)){
				inst->Internal.Idx = GetIndex(&inst->SelectedElem);

				if(inst->Internal.Idx != inst->Internal.LastIdx){
					//We've changed indecies need to head back to init to reset the sh status
					inst->Valid = FALSE;
					inst->Internal.Fbs.ShGetInfo.Enable = FALSE;

					inst->Internal.State = tmSH_CONTROL_INIT;
				}
				else{
					//Here we can start parsing commands
					if(inst->ElasticMoveAbs){
						//Setup the elastic move absolute block and execute it
						inst->Internal.Fbs.ElMoveAbs.Axis = &inst->Internal.CurrentAxis;
						inst->Internal.Fbs.ElMoveAbs.Position = inst->Parameters->Position;
						inst->Internal.Fbs.ElMoveAbs.Velocity = inst->Parameters->Vel;
						inst->Internal.Fbs.ElMoveAbs.Acceleration = inst->Parameters->Accel;
						inst->Internal.Fbs.ElMoveAbs.Deceleration = inst->Parameters->Decel;

						inst->Internal.Fbs.ElMoveAbs.Execute = TRUE;

						inst->Internal.State = tmSH_CONTROL_EL_MOVE_ABS;
					}
					else if(inst->ElasticMoveAdd){
						//Setup the elastic move additve block and execute it
						inst->Internal.Fbs.ElMoveAdd.Axis = &inst->Internal.CurrentAxis;
						inst->Internal.Fbs.ElMoveAdd.Distance = inst->Parameters->Distance;
						inst->Internal.Fbs.ElMoveAdd.Velocity = inst->Parameters->Vel;
						inst->Internal.Fbs.ElMoveAdd.Acceleration = inst->Parameters->Accel;
						inst->Internal.Fbs.ElMoveAdd.Deceleration = inst->Parameters->Decel;

						inst->Internal.Fbs.ElMoveAdd.Execute = TRUE;

						inst->Internal.State = tmSH_CONTROL_EL_MOVE_ADD;
					}//End of commands check conditionals
				}
			}
			else{//We've received an invalid selection, need to reset the flags and Sh Status
				inst->Valid = FALSE;
				inst->Internal.Fbs.ShGetInfo.Enable = FALSE;

				inst->Internal.State = tmSH_CONTROL_INIT;
			}

			break;
		case tmSH_CONTROL_EL_MOVE_ABS:
			//******************************************************************************** Elastic Move absolute state
			if(inst->Internal.Fbs.ElMoveAbs.Error){
				inst->Error = TRUE;
				inst->ErrorID = tmSH_CONTROL_ERR_EL_MOVE;

				inst->Internal.State = tmSH_CONTROL_ERROR;
			}
			else if(inst->Internal.Fbs.ElMoveAbs.Active){
				inst->MovementActive = TRUE;
			}
			else if(inst->Internal.Fbs.ElMoveAbs.Done){
				inst->Internal.Fbs.ElMoveAbs.Execute = FALSE;
				inst->MovementActive = FALSE;
				inst->MovementDone = TRUE;

				inst->Internal.State = tmSH_CONTROL_MOVE_DONE;
			}
			break;
		case tmSH_CONTROL_EL_MOVE_ADD:
			//******************************************************************************** Elastic Move Additive state
			if(inst->Internal.Fbs.ElMoveAdd.Error){
				inst->Error = TRUE;
				inst->ErrorID = tmSH_CONTROL_ERR_EL_MOVE;

				inst->Internal.State = tmSH_CONTROL_ERROR;
			}
			else if(inst->Internal.Fbs.ElMoveAdd.Done){
				inst->MovementActive = FALSE;
				inst->MovementDone = TRUE;

				inst->Internal.Fbs.ElMoveAdd.Execute = FALSE;

				inst->Internal.State = tmSH_CONTROL_MOVE_DONE;
			}
			else{
				inst->MovementActive = TRUE;
			}
			break;
		case tmSH_CONTROL_MOVE_DONE:
			//******************************************************************************** Movement Done State
			if(!inst->ElasticMoveAbs
				&& !inst->ElasticMoveAdd){
				inst->MovementDone = FALSE;

				inst->Internal.State = tmSH_CONTROL_IDLE;
			}
			break;
		case tmSH_CONTROL_ERROR:
			//******************************************************************************** Error State
			if(!inst->Enable){
				inst->Error = FALSE;
				inst->ErrorID = tmSH_CONTROL_ERR_OK;

				inst->Internal.Fbs.ElMoveAbs.Execute = FALSE;
				inst->Internal.Fbs.ElMoveAdd.Execute = FALSE;
				inst->Internal.Fbs.ShGetInfo.Enable = FALSE;

				inst->Internal.Idx = 0;
				inst->Internal.LastIdx = 0;

				inst->Internal.State = tmSH_CONTROL_OFF;
			}
			break;
	}
	//FB calls

	MC_BR_ShReadInfo_AcpTrak(&inst->Internal.Fbs.ShGetInfo);
	MC_BR_ElasticMoveAbs_AcpTrak(&inst->Internal.Fbs.ElMoveAbs);
	MC_BR_ElasticMoveAdd_AcpTrak(&inst->Internal.Fbs.ElMoveAdd);
}
```

- Visualisation Logical/mappView (not shown)

### Program Logical/Source/TrackMaster (ANSIC)

#### Cyclic.c - Cyclic code
```c
/*********************************************************************************
 * Copyright: B&R Industrial Automation GmbH
 * Author:    trostelc
 * Created:   October 16, 2020/5:04 PM
 *********************************************************************************/

#include <bur/plctypes.h>

#ifdef _DEFAULT_INCLUDES
#include <AsDefault.h>
#endif

void _CYCLIC ProgramCyclic(void)
{
	//Build the SVG transform string
	//Start by adding the svg viewbox
	//Loop through the shuttle mon, if the shuttle is enabled, you'll take the X/Y/Z/rot and use it to build a <g> in the svg

	switch (state){
		case 0:
			if(start || gPowered){
				TrackMasterCore.Assembly = &gAssembly_1;
				TrackMasterCore.ShuttleMon = &gShuttleMon;
				TrackMasterCore.Enable = 1;

				//Set parameters for View box (this comes from the automatically generated SVG)
				TrackMasterCore.ViewBoxCfg.MinX = -3.37558;
				TrackMasterCore.ViewBoxCfg.MinY = -0.745;
				TrackMasterCore.ViewBoxCfg.Width = 4.11115;
				TrackMasterCore.ViewBoxCfg.Height = 0.86;

				state = 10;
			}
			break;
		case 10:
			if(TrackMasterCore.Active){
				ShControl.Enable = 1;
				ShControl.Handle = TrackMasterCore.Handle;
				ShControl.Parameters = &shPars;

				state = 20;
			}
			break;
		case 20:
			break;

	}

	brdkStrCpy(&ShControl.SelectedElem,&selectedId);

	tmCore(&TrackMasterCore);
	tmShuttleControl(&ShControl);

	//GetIndex();
}
```

#### Init.c - Initialization code
```c
#include <bur/plctypes.h>

#ifdef _DEFAULT_INCLUDES
	#include <AsDefault.h>
#endif

void _INIT ProgramInit(void)
{
	brsmemset(&selectedId,0,sizeof(selectedId));
	shPars.Accel = 10;
	shPars.Decel = 10;
	shPars.Vel = 1;
	coreOptions.Color.Enabled = 1;
	coreOptions.Color.Offsets.Red = 0;
	coreOptions.Color.Offsets.Green = 1;
	coreOptions.Color.Offsets.Blue = 2;
	TrackMasterCore.Options = &coreOptions;
}
```

#### Variables.var - Local variables
```iecst
VAR
	selectedId : STRING[80];
	Selected : BOOL;
	TrackMasterCore : tmCore;
	ShControl : tmShuttleControl;
	shPars : tmShuttleControlParsTyp;
	state : USINT;
	start : BOOL;
	coreOptions : tmCoreOptionsTyp;
END_VAR
```

### Program Logical/Source/Trak/TrakMain (ANSIC)

#### Variables.var
```iecst
VAR
	axis : McAxisType;
	asmPowerOn : MC_BR_AsmPowerOn_AcpTrak;
	state : USINT;
	secAddShuttle : MC_BR_SecAddShuttle_AcpTrak;
	routedMoveVel : MC_BR_RoutedMoveVel_AcpTrak;
	secGetShuttle : MC_BR_SecGetShuttle_AcpTrak;
	start : BOOL;
	SendCmd : BOOL;
	count : USINT;
	maxShuttle : USINT;
	copyUserData : MC_BR_ShCopyUserData_AcpTrak;
	userData : UserDataTyp;
END_VAR
```

#### Cyclic.c
```c
#include <bur/plctypes.h>

#ifdef _DEFAULT_INCLUDES
	#include <AsDefault.h>
#endif

void _CYCLIC ProgramCyclic(void)
{
	switch (state){
		case 0:
			if(start){
				asmPowerOn.Assembly = &gAssembly_1;
				asmPowerOn.Execute = 1;

				state = 10;
			}
			break;
		case 10:
			if(asmPowerOn.Done){
				secAddShuttle.Execute = 1;
				secAddShuttle.Sector = &secMain;
				secAddShuttle.Position = 0;

				state = 20;
			}
			break;
		case 20:
			if(secAddShuttle.Done){
				secAddShuttle.Execute = 0;

				if(count < 1){
					state = 21;
					secAddShuttle.Position = 0.5;
					count++;
				}
				else{
					state = 30;
				}
			}
			break;
		case 21:
			secAddShuttle.Execute = 1;
			state = 20;
			break;
		case 30:
			gPowered = 1;

			break;
	}
	MC_BR_AsmPowerOn_AcpTrak(&asmPowerOn);
	MC_BR_SecAddShuttle_AcpTrak(&secAddShuttle);
	MC_BR_RoutedMoveVel_AcpTrak(&routedMoveVel);

}
```

#### Init.c
```c
#include <bur/plctypes.h>

#ifdef _DEFAULT_INCLUDES
	#include <AsDefault.h>
#endif

void _INIT ProgramInit(void)
{
	maxShuttle = 5;
}
```

### Program Logical/Source/Program

#### Variables.var
```iecst
VAR
	selectedId : STRING[80];
	Selected : BOOL;
	TrackMasterCore : tmCore;
	ShControl : tmShuttleControl;
	shPars : tmShuttleControlParsTyp;
END_VAR
```

#### Cyclic.c
```c
/*********************************************************************************
 * Copyright: B&R Industrial Automation GmbH
 * Author:    trostelc
 * Created:   October 16, 2020/5:04 PM
 *********************************************************************************/

#include <bur/plctypes.h>

#ifdef _DEFAULT_INCLUDES
#include <AsDefault.h>
#endif
void BuildStr(){
	LREAL width;
	LREAL length;
	width = gShuttleMon.Shuttle[idx].Width / 1000.0;
	length = (gShuttleMon.Shuttle[idx].ExtentToBack + gShuttleMon.Shuttle[idx].ExtentToFront)/ 1000.0;

	snprintf2(tmp,150,"<g id=\"Shuttle\">");
	brsstrcat(&svgContent,&tmp);

	snprintf2(tmp,150,"<polygon id=\"box\" x=\"%f\" y=\"%f\" points=\"0,0 %0f,0 , %f,%f %f,%f 0,%f\" style=\"fill:rgb(0,255,0);\"/>",
		-gShuttleMon.Shuttle[idx].ExtentToBack / 1000.0,
		-width,
		(length-width/2.0),
		length,
		width/2.0,
		(length-width/2.0),
		width,
		width);
	brsstrcat(&svgContent,&tmp);

	snprintf2(tmp,150,"<text x=\"%f\" y=\"%f\" font-weight=\"bold\" font-size=\"0.035px\">%d</text>",
		length * 0,
		width * 3.0 / 4.0,
		gShuttleMon.Shuttle[idx].Index);
	brsstrcat(&svgContent,&tmp);

	//Create an invisible bounding rectangle to handle the click event. "Invisible" by using the alpha channel, if you use the
	//Vibisility property, the click event will not fire for the SVG
	snprintf2(tmp,150,"<rect id=\"ID%d\" width=\".05\" height=\"0.05\" style=\"fill:rgba(0,0,255,0)\"/>",
		gShuttleMon.Shuttle[idx].Index,
		length ,
		width);
	brsstrcat(&svgContent,&tmp);

	brsstrcat(&svgContent,&"</g>");
}
void GetIndex(){
	char buf[2];
	//Get a substring of the first 3 characters
	brdkStrSubStr(&buf,&selectedId,0,3);
	//Look at the start of the selectedID, if it starts with #ID then we know a shuttle has been clicked
	if(0 == brsstrcmp(&buf,&"#ID")){
		Selected = 1;
	}
	else{
		Selected = 0;
	}
}
void _CYCLIC ProgramCyclic(void)
{
	//Build the SVG transform string
	//Start by adding the svg viewbox
	//Loop through the shuttle mon, if the shuttle is enabled, you'll take the X/Y/Z/rot and use it to build a <g> in the svg

	if(testEnable){
		//Reset the entire SVG additional content
		brsmemset(&svgContent,0,sizeof(svgContent));
		brsmemset(&svgTransform,0,sizeof(svgTransform));

		brsstrcat(&svgContent,&"<svg viewBox=\"-3.37558 -0.745 4.11115 0.86\">");
		for (idx = 0; idx < 9; idx++){
			if(gShuttleMon.Shuttle[idx].Available){

				BuildStr();

				snprintf2(tmp,150,"[{\"select\":\"#Shuttle\",\"duration\":100,\"display\":true,\"translate\":[%f,%f]}]",
					gShuttleMon.Shuttle[idx].Position.X / 1000.0 - gShuttleMon.Shuttle[idx].ExtentToBack / 1000.0,
					-gShuttleMon.Shuttle[idx].Position.Y / 1000.0 - gShuttleMon.Shuttle[idx].Width / 2000.0);
				brsstrcat(&svgTransform,&tmp);

			}
		}
		brsstrcat(&svgContent,&"</svg>");
	}
	GetIndex();
}
```

#### Init.c
```c
#include <bur/plctypes.h>

#ifdef _DEFAULT_INCLUDES
	#include <AsDefault.h>
#endif

void _INIT ProgramInit(void)
{
	brsmemset(&svgContent,0,sizeof(svgContent));
	brsmemset(&svgTransform,0,sizeof(svgTransform));
	brsmemset(&selectedId,0,sizeof(selectedId));
}
```

- Version.bat (not shown)

### Program Logical/Source/Support/Version/Version (IEC)

#### Version.st - Init, cyclic, exit code
```iecst
PROGRAM _CYCLIC
Version := '99d5fba';
Author := 'BRGLOBAL\trostelc';
Date := '';
END_PROGRAM
```

#### Variables.var - Local variables
```iecst
VAR
	Version : STRING[255]; (*Revision Number of the commit*)
	Author : STRING[255]; (*Author of the commit*)
	Date : STRING[255]; (*Date of the commit*)
END_VAR
```

### Program Logical/Source/Support/MachineInfo (IEC)

#### Init.st - Init code
```iecst
PROGRAM _INIT
	MachineLastRevisionDate;
	MachineSoftwareVersion;

END_PROGRAM
```

#### Variables.var - Local variables
```iecst
VAR
	MachineSoftwareVersion : STRING[80] := '* Dev-0.0.1-9-a71ff01';
	MachineLastRevisionDate : DATE_AND_TIME := DT#2020-11-11-17:07;
END_VAR
```

- gAssembly_1.wsp (not shown)

Listed in the project but not available here: Logical/Libraries/brdkSTR/brdkSTR.typ, Logical/Libraries/brdkSTR/brdkSTR.var, Logical/Libraries/brdkSTR/brdkSTR.fun, Logical/Libraries/brdkSTR/brdkStrAppendUdintToA.c, Logical/Libraries/brdkSTR/brdkStrAToDint.c, Logical/Libraries/brdkSTR/brdkStrAToUdint.c, Logical/Libraries/brdkSTR/brdkStrCat.c, Logical/Libraries/brdkSTR/brdkStrCatAtChar.c, Logical/Libraries/brdkSTR/brdkStrCharAt.c, Logical/Libraries/brdkSTR/brdkStrCharCount.c, Logical/Libraries/brdkSTR/brdkStrCmp.c, Logical/Libraries/brdkSTR/brdkStrCpy.c, Logical/Libraries/brdkSTR/brdkStrCrc32.c, Logical/Libraries/brdkSTR/brdkStrDintToA.c, Logical/Libraries/brdkSTR/brdkStrFill.c, Logical/Libraries/brdkSTR/brdkStrIndexOf.c, Logical/Libraries/brdkSTR/brdkStrInsertAtPos.c, Logical/Libraries/brdkSTR/brdkStrLen.c, Logical/Libraries/brdkSTR/brdkStrMemCmp.c, Logical/Libraries/brdkSTR/brdkStrMemCpy.c, Logical/Libraries/brdkSTR/brdkStrMemMove.c, Logical/Libraries/brdkSTR/brdkStrMemSet.c, Logical/Libraries/brdkSTR/brdkStrMove.c, Logical/Libraries/brdkSTR/brdkStrNCpy.c, Logical/Libraries/brdkSTR/brdkStrRemove.c, Logical/Libraries/brdkSTR/brdkStrRepeat.c, Logical/Libraries/brdkSTR/brdkStrReplace.c, Logical/Libraries/brdkSTR/brdkStrReverse.c, Logical/Libraries/brdkSTR/brdkStrReverseWords.c, Logical/Libraries/brdkSTR/brdkStrSearch.c, Logical/Libraries/brdkSTR/brdkStrSlice.c, Logical/Libraries/brdkSTR/brdkStrSubStr.c, Logical/Libraries/brdkSTR/brdkStrToDec.c, Logical/Libraries/brdkSTR/brdkStrToHex.c, Logical/Libraries/brdkSTR/brdkStrToLowerCase.c, Logical/Libraries/brdkSTR/brdkStrToUpperCase.c, Logical/Libraries/brdkSTR/brdkStrToUpperCaseWords.c, Logical/Libraries/brdkSTR/brdkStrTrim.c, Logical/Libraries/brdkSTR/brdkStrUdintToA.c, Logical/Libraries/brdkSTR/brdkSTR_func.h, Logical/Libraries/brdkSTR/brdkSTR_func.c, Logical/Source/TrackMaster/Exit.c, Logical/Source/TrackMaster/Types.typ, Logical/Source/Support/Version/Version/Types.typ, Logical/Source/Support/MachineInfo/Cyclic.st, Logical/Source/Support/MachineInfo/Exit.st, Logical/Source/Support/MachineInfo/Types.typ
